KUKA KRL program: chk_w8_tools_ok.src, chk_w8_tools_ok.dat

--- chk_w8_tools_ok.src ---
&ACCESS RVO4
&COMMENT Checagem das ferramentas nos docks
DEF chk_w8_tools_ok( )
;Routine to check all dock stations before take the tool
;Please, verify the inputs to each robot
;Verificar as entradas para adaptar à cada robô
;Dock 1 - 161
;Dock 2 - 169
;Dock 3 - 177
;Dock 4 - 185
;Dock 5 - 193
;Dock 6 - 201
;Dock 7 - 209

$TIMER[10] = 0
$TIMER_STOP[10] = FALSE

wait for (( $in[161]) and ($IN[169]) and ($IN[177]) and ($IN[185]) and ($in[193]) and ($in[201]) and ($in[209]))

$TIMER_STOP[10] = TRUE
$TIMER[10] = 0

END

--- chk_w8_tools_ok.dat ---
&ACCESS RVO4
&COMMENT Checagem das ferramentas nos docks
DEFDAT chk_w8_tools_ok PUBLIC
ENDDAT
